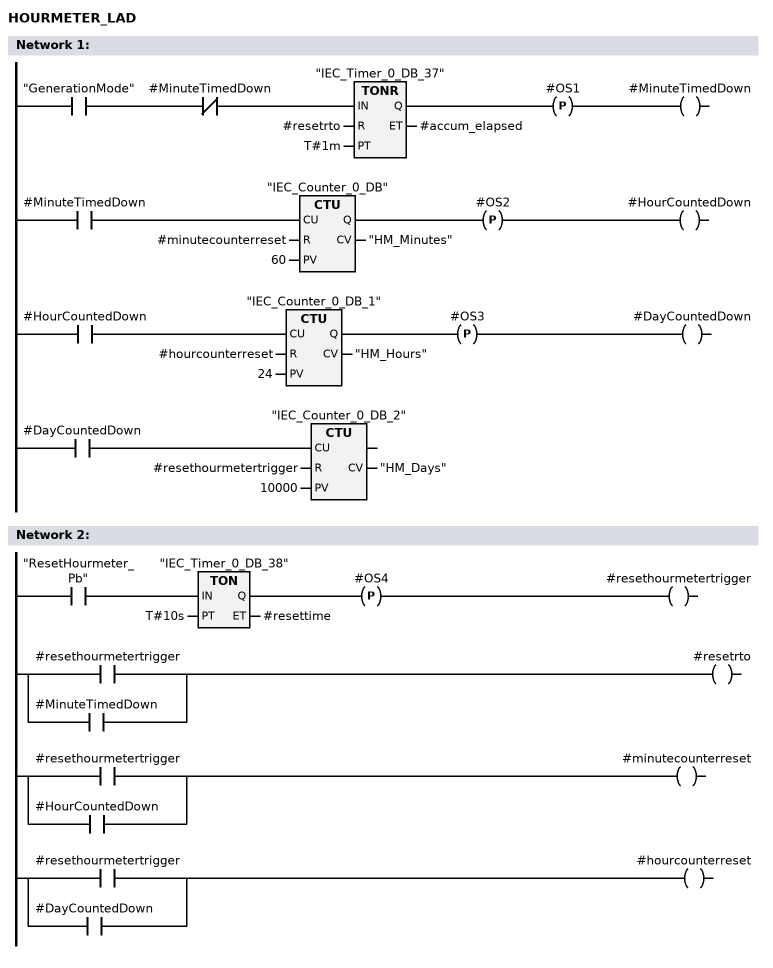
   "IEC_Timer_0_DB_37".TONR(IN := "GenerationMode" AND NOT #MinuteTimedDown,
                           R := #resetrto,
                           PT := T#1m,
                           ET => #accum_elapsed);
   #_w1 := "IEC_Timer_0_DB_37".Q AND NOT #OS1;   // rising edge
   #OS1 := "IEC_Timer_0_DB_37".Q;
   #MinuteTimedDown := #_w1;
   "IEC_Counter_0_DB".CTU(CU := #MinuteTimedDown, R := #minutecounterreset, PV := 60, CV => "HM_Minutes");
   #_w2 := "IEC_Counter_0_DB".Q AND NOT #OS2;   // rising edge
   #OS2 := "IEC_Counter_0_DB".Q;
   #HourCountedDown := #_w2;
   "IEC_Counter_0_DB_1".CTU(CU := #HourCountedDown, R := #hourcounterreset, PV := 24, CV => "HM_Hours");
   #_w3 := "IEC_Counter_0_DB_1".Q AND NOT #OS3;   // rising edge
   #OS3 := "IEC_Counter_0_DB_1".Q;
   #DayCountedDown := #_w3;
   "IEC_Counter_0_DB_2".CTU(CU := #DayCountedDown, R := #resethourmetertrigger, PV := 10000, CV => "HM_Days");
END_REGION

REGION Network 2
   "IEC_Timer_0_DB_38".TON(IN := "ResetHourmeter_Pb", PT := T#10s, ET => #resettime);
   #_w1 := "IEC_Timer_0_DB_38".Q AND NOT #OS4;   // rising edge
   #OS4 := "IEC_Timer_0_DB_38".Q;
   #resethourmetertrigger := #_w1;
   #resetrto := #resethourmetertrigger OR #MinuteTimedDown;
   #minutecounterreset := #resethourmetertrigger OR #HourCountedDown;
   #hourcounterreset := #resethourmetertrigger OR #DayCountedDown;
END_REGION
END_FUNCTION_BLOCK

FUNCTION_BLOCK "HOURMETER_FBD"   // FB20, FBD
{ S7_Optimized_Access := 'TRUE' }
VERSION : 0.1
   VAR
      OS1 : Bool;
      OS2 : Bool;
      OS3 : Bool;
      OS4 : Bool;
      rtotimerreset : Bool;
      minutecounterreset : Bool;
      hourcounterreset : Bool;
      hourmeterresettrigger : Bool;
      accumulatedtime : Time;
      minutetimeddown : Bool;
      hourcounteddown : Bool;
      daycounteddown : Bool;
   END_VAR
   VAR_TEMP   // added for the SCL form of the ladder/FBD networks
      _w1 : Bool;
      _w2 : Bool;
      _w3 : Bool;
   END_VAR
BEGIN

REGION Network 1
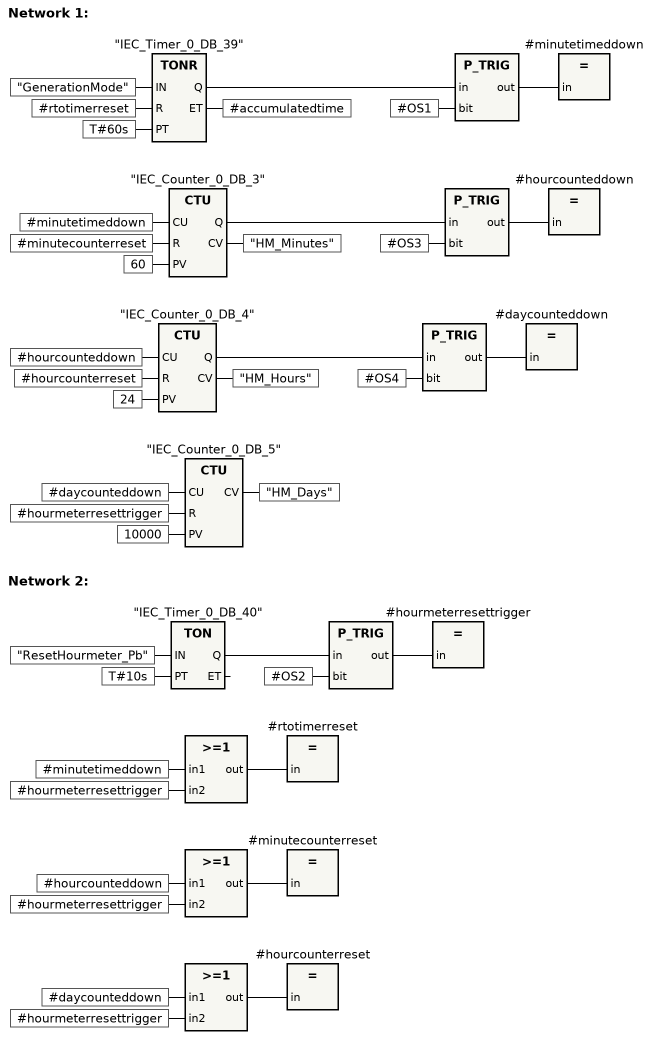
   "IEC_Timer_0_DB_39".TONR(IN := "GenerationMode", R := #rtotimerreset, PT := T#60s, ET => #accumulatedtime);
   #_w1 := "IEC_Timer_0_DB_39".Q AND NOT #OS1;   // rising edge
   #OS1 := "IEC_Timer_0_DB_39".Q;
   #minutetimeddown := #_w1;
   "IEC_Counter_0_DB_3".CTU(CU := #minutetimeddown, R := #minutecounterreset, PV := 60, CV => "HM_Minutes");
   #_w2 := "IEC_Counter_0_DB_3".Q AND NOT #OS3;   // rising edge
   #OS3 := "IEC_Counter_0_DB_3".Q;
   #hourcounteddown := #_w2;
   "IEC_Counter_0_DB_4".CTU(CU := #hourcounteddown, R := #hourcounterreset, PV := 24, CV => "HM_Hours");
   #_w3 := "IEC_Counter_0_DB_4".Q AND NOT #OS4;   // rising edge
   #OS4 := "IEC_Counter_0_DB_4".Q;
   #daycounteddown := #_w3;
   "IEC_Counter_0_DB_5".CTU(CU := #daycounteddown, R := #hourmeterresettrigger, PV := 10000, CV => "HM_Days");
END_REGION

REGION Network 2
   "IEC_Timer_0_DB_40".TON(IN := "ResetHourmeter_Pb", PT := T#10s);
   #_w1 := "IEC_Timer_0_DB_40".Q AND NOT #OS2;   // rising edge
   #OS2 := "IEC_Timer_0_DB_40".Q;
   #hourmeterresettrigger := #_w1;
   #rtotimerreset := #minutetimeddown OR #hourmeterresettrigger;
   #minutecounterreset := #hourcounteddown OR #hourmeterresettrigger;
   #hourcounterreset := #daycounteddown OR #hourmeterresettrigger;
END_REGION
END_FUNCTION_BLOCK

FUNCTION_BLOCK "HOURMETER_SCL"   // FB21, SCL
{ S7_Optimized_Access := 'TRUE' }
VERSION : 0.1
   VAR
      rtotimerreset : Bool;
      minutecounterreset : Bool;
      hourcounterreset : Bool;
      hourmeterresettrigger : Bool;
      accumulatedtime : Time;
      minutetimeddown : Bool;
      hourcounteddown : Bool;
      daycounteddown : Bool;
   END_VAR
BEGIN
   IF "GenerationMode" THEN
       "IEC_Timer_0_DB_41".TONR(IN := TRUE,
                                R := #rtotimerreset,
                                PT := T#60s,
                                Q => #minutetimeddown,
                                ET => #accumulatedtime);
   END_IF;

   IF #minutetimeddown THEN
       RESET_TIMER("IEC_Timer_0_DB_41");
   END_IF;

   "IEC_Counter_0_DB_6".CTU(CU:=#minutetimeddown,
                            R:=#minutecounterreset,
                            PV:=60,
                            Q=>#hourcounteddown,
                            CV=>"HM_Minutes");

   "IEC_Counter_0_DB_7".CTU(CU:=#hourcounteddown,
                            R:=#hourcounterreset,
                            PV:=24,
                            Q=>#daycounteddown,
                            CV=>"HM_Hours");

   "IEC_Counter_0_DB_9".CTU(CU:=#daycounteddown,
                            R:=#hourmeterresettrigger,
                            PV:=10000,
                            CV=>"HM_Days");

   IF "ResetHourmeter_Pb" THEN
       "IEC_Timer_0_DB_42".TON(IN:=TRUE,
                               PT:=T#10s,
                               Q=>#hourmeterresettrigger);
   ELSE
       RESET_TIMER("IEC_Timer_0_DB_42");
   END_IF;

   IF #hourmeterresettrigger OR #minutetimeddown THEN
       #rtotimerreset := 1;
   ELSE
       #rtotimerreset := 0;
   END_IF;

   IF #hourmeterresettrigger OR #hourcounteddown THEN
       #minutecounterreset := 1;
   ELSE
       #minutecounterreset := 0;
   END_IF;

   IF #hourmeterresettrigger OR #daycounteddown THEN
       #hourcounterreset := 1;
   ELSE
       #hourcounterreset := 0;
   END_IF;
END_FUNCTION_BLOCK

FUNCTION_BLOCK "HOURMETER_STL"   // FB22, STL
{ S7_Optimized_Access := 'TRUE' }
VERSION : 0.1
   VAR
      hourmeterresettrigger : Bool;
      minutecounterreset : Bool;
      hourcounterreset : Bool;
      minutetimeddown : Bool;
      hourcounteddown : Bool;
      daycounteddown : Bool;
      accumulatedtime : Time;
      rtotimerreset : Bool;
   END_VAR
   VAR_TEMP
      toomanydays : Bool;
      acctime : Time;
   END_VAR
BEGIN

REGION Network 1
         A     "GenerationMode";
         JC    RTOtimer;
         CLR;
         JU    EndOfLine;

   RTOtimer:CALL  TONR, "IEC_Timer_0_DB_43"
         ( IN := TRUE,
           R  := #rtotimerreset,
           PT := T#1m,
           Q  := #minutetimeddown,
           ET := #accumulatedtime
         );

         CALL  CTU, "IEC_Counter_0_DB_10"
         ( CU := #minutetimeddown,
           R  := #minutecounterreset,
           PV := 60,
           Q  := #hourcounteddown,
           CV := "HM_Minutes"
         );

         CALL  CTU, "IEC_Counter_0_DB_11"
         ( CU := #hourcounteddown,
           R  := #hourcounterreset,
           PV := 24,
           Q  := #daycounteddown,
           CV := "HM_Hours"
         );

         CALL  CTU, "IEC_Counter_0_DB_12"
         ( CU := #daycounteddown,
           R  := #hourmeterresettrigger,
           PV := 10000,
           Q  := #toomanydays,
           CV := "HM_Days"
         );

         JU    ResetEvaluate;

   ResetEvaluate:CLR;
         A     "ResetHourmeter_Pb";
         JC    ResetHourmeter;
         CALL  RESET_TIMER
         ( "TIMER" := "IEC_Timer_0_DB_44"
         );
         JU    EndOfLine;

   ResetHourmeter:CALL  TON, "IEC_Timer_0_DB_44"
         ( IN := TRUE,
           PT := T#10s,
           Q  := #hourmeterresettrigger,
           ET := #acctime
         );


   EndOfLine:A     #hourmeterresettrigger;
         O     #minutetimeddown;
         =     #rtotimerreset;
         CLR;
         A     #hourmeterresettrigger;
         O     #hourcounteddown;
         =     #minutecounterreset;
         CLR;
         A     #hourmeterresettrigger;
         O     #daycounteddown;
         =     #hourcounterreset;
         CLR;
         NOT;
         R     #hourmeterresettrigger;
END_REGION
END_FUNCTION_BLOCK

FUNCTION "SCP" : Void   // FC1, FBD
{ S7_Optimized_Access := 'TRUE' }
VERSION : 0.1
   VAR_INPUT
      Input_Min : Int;
      Input_Signal : Int;
      Input_Max : Int;
      Output_Min : Int;
      Output_Max : Int;
   END_VAR
   VAR_OUTPUT
      SV : Int;
   END_VAR
   VAR_TEMP
      tv : Real;
   END_VAR
BEGIN

REGION Network 1
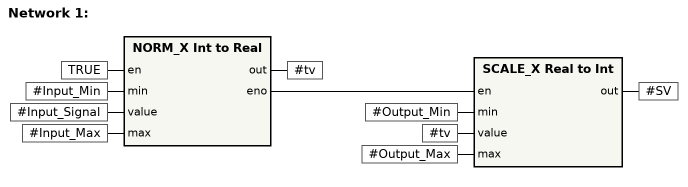
   IF TRUE THEN
       #tv := NORM_X(MIN := #Input_Min, VALUE := #Input_Signal, MAX := #Input_Max);
       #SV := SCALE_X(MIN := #Output_Min, VALUE := #tv, MAX := #Output_Max);
   END_IF;
END_REGION
END_FUNCTION

FUNCTION "CONVERTTIME" : Void   // FC2, FBD
{ S7_Optimized_Access := 'TRUE' }
VERSION : 0.1
   VAR_INPUT
      Int1 : Int;
   END_VAR
   VAR_OUTPUT
      Time1 : Time;
   END_VAR
   VAR_TEMP
      tv : Int;
   END_VAR
BEGIN

REGION Network 1
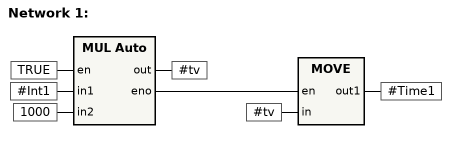
   IF TRUE THEN
       #tv := #Int1 * 1000;
       #Time1 := #tv;
   END_IF;
END_REGION
END_FUNCTION

ORGANIZATION_BLOCK "Main"   // OB1, LAD, ProgramCycle
TITLE = "Main Program Sweep (Cycle)"
{ S7_Optimized_Access := 'TRUE' }
VERSION : 0.1
   VAR_INPUT
      Initial_Call : Bool;   // Initial call of this OB
      Remanence : Bool;   // =True, if remanent data are available
   END_VAR
   VAR_TEMP
      SequenceInit : Bool;
      InitSequence : Bool;
   END_VAR
   VAR_TEMP   // added for the SCL form of the ladder/FBD networks
      _w1 : Bool;
      _w2 : Bool;
      _w3 : Bool;
      _w4 : Bool;
   END_VAR
BEGIN

REGION Network 1
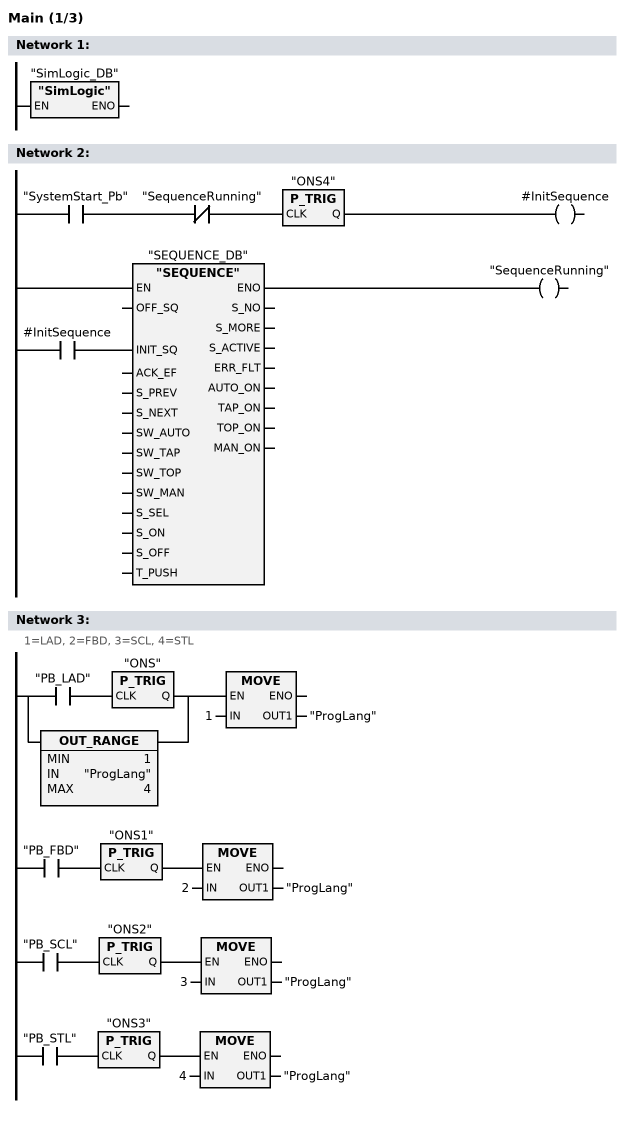
   RUNG wire#powerrail
      "SimLogic_DB"()
   END_RUNG
   // the same network as SCL:
   "SimLogic_DB"();   // "SimLogic"
END_REGION

REGION Network 2
   RUNG wire#powerrail
      Contact( "SystemStart_Pb" )
      I_Contact( "SequenceRunning" )
      P_Trig( "ONS4" )
      Coil( #InitSequence )
   END_RUNG
   RUNG wire#powerrail
      "SEQUENCE_DB"(INIT_SQ := wire#w1, OFF_SQ :=, ACK_EF :=, S_PREV :=, S_NEXT :=, SW_AUTO :=, SW_TAP :=, SW_TOP :=, SW_MAN :=, S_SEL :=, S_ON :=, S_OFF :=, T_PUSH :=, S_NO =>, S_MORE =>, S_ACTIVE =>, ERR_FLT =>, AUTO_ON =>, TAP_ON =>, TOP_ON =>, MAN_ON =>)
      Coil( "SequenceRunning" )
   END_RUNG
   RUNG wire#powerrail
      Contact( #InitSequence )
   END_RUNG wire#w1
   // the same network as SCL:
   #_w1 := "SystemStart_Pb" AND NOT "SequenceRunning";
   #_w2 := #_w1 AND NOT "ONS4";   // rising edge
   "ONS4" := #_w1;
   #InitSequence := #_w2;
   "SEQUENCE_DB"(INIT_SQ := #InitSequence, ENO => #_w3);   // "SEQUENCE"
   "SequenceRunning" := #_w3;
END_REGION

REGION Network 3
   // 1=LAD, 2=FBD, 3=SCL, 4=STL
   #_w1 := "PB_LAD" AND NOT "ONS";   // rising edge
   "ONS" := "PB_LAD";
   IF #_w1 OR ("ProgLang" < 1) OR ("ProgLang" > 4) THEN "ProgLang" := 1; END_IF;
   #_w2 := "PB_FBD" AND NOT "ONS1";   // rising edge
   "ONS1" := "PB_FBD";
   IF #_w2 THEN "ProgLang" := 2; END_IF;
   #_w3 := "PB_SCL" AND NOT "ONS2";   // rising edge
   "ONS2" := "PB_SCL";
   IF #_w3 THEN "ProgLang" := 3; END_IF;
   #_w4 := "PB_STL" AND NOT "ONS3";   // rising edge
   "ONS3" := "PB_STL";
   IF #_w4 THEN "ProgLang" := 4; END_IF;
END_REGION

REGION Network 4
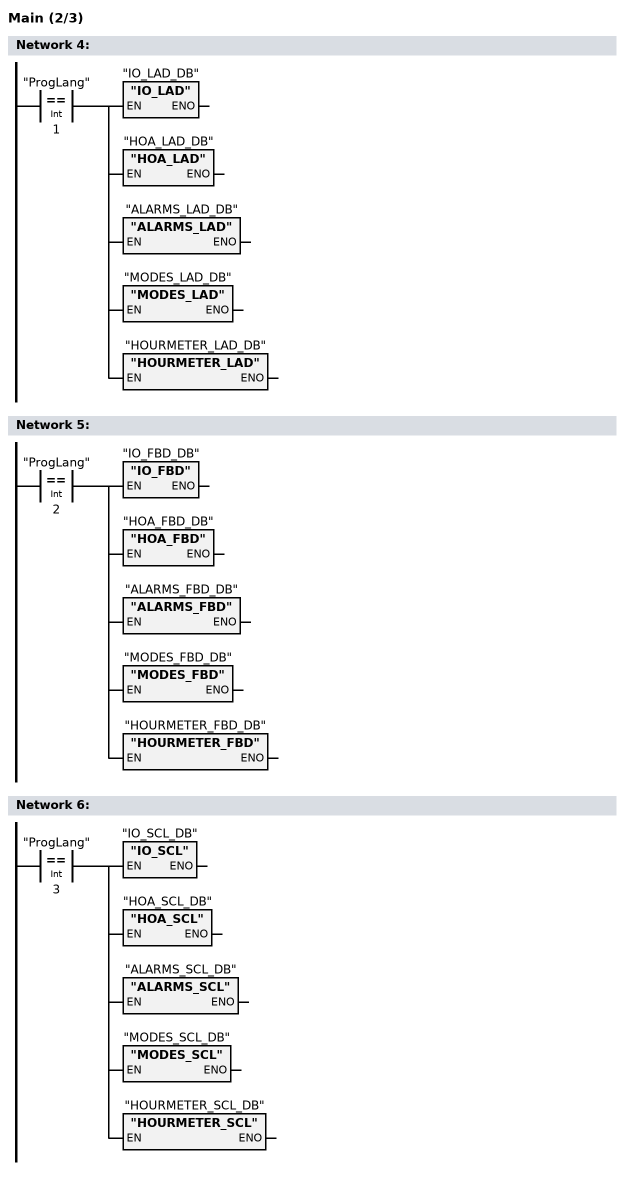
   RUNG wire#powerrail
      { S7_Templates := "SrcType := Int" } EQ_Contact(in1 := "ProgLang", in2 := 1)
      wire#w1
      "IO_LAD_DB"()
   END_RUNG
   RUNG wire#w1
      "HOA_LAD_DB"()
   END_RUNG
   RUNG wire#w1
      "ALARMS_LAD_DB"()
   END_RUNG
   RUNG wire#w1
      "MODES_LAD_DB"()
   END_RUNG
   RUNG wire#w1
      "HOURMETER_LAD_DB"()
   END_RUNG
   // the same network as SCL:
   #_w1 := "ProgLang" = 1;
   IF #_w1 THEN
       "IO_LAD_DB"();   // "IO_LAD"
       "HOA_LAD_DB"();   // "HOA_LAD"
       "ALARMS_LAD_DB"();   // "ALARMS_LAD"
       "MODES_LAD_DB"();   // "MODES_LAD"
       "HOURMETER_LAD_DB"();   // "HOURMETER_LAD"
   END_IF;
END_REGION

REGION Network 5
   RUNG wire#powerrail
      { S7_Templates := "SrcType := Int" } EQ_Contact(in1 := "ProgLang", in2 := 2)
      wire#w1
      "IO_FBD_DB"()
   END_RUNG
   RUNG wire#w1
      "HOA_FBD_DB"()
   END_RUNG
   RUNG wire#w1
      "ALARMS_FBD_DB"()
   END_RUNG
   RUNG wire#w1
      "MODES_FBD_DB"()
   END_RUNG
   RUNG wire#w1
      "HOURMETER_FBD_DB"()
   END_RUNG
   // the same network as SCL:
   #_w1 := "ProgLang" = 2;
   IF #_w1 THEN
       "IO_FBD_DB"();   // "IO_FBD"
       "HOA_FBD_DB"();   // "HOA_FBD"
       "ALARMS_FBD_DB"();   // "ALARMS_FBD"
       "MODES_FBD_DB"();   // "MODES_FBD"
       "HOURMETER_FBD_DB"();   // "HOURMETER_FBD"
   END_IF;
END_REGION

REGION Network 6
   RUNG wire#powerrail
      { S7_Templates := "SrcType := Int" } EQ_Contact(in1 := "ProgLang", in2 := 3)
      wire#w1
      "IO_SCL_DB"()
   END_RUNG
   RUNG wire#w1
      "HOA_SCL_DB"()
   END_RUNG
   RUNG wire#w1
      "ALARMS_SCL_DB"()
   END_RUNG
   RUNG wire#w1
      "MODES_SCL_DB"()
   END_RUNG
   RUNG wire#w1
      "HOURMETER_SCL_DB"()
   END_RUNG
   // the same network as SCL:
   #_w1 := "ProgLang" = 3;
   IF #_w1 THEN
       "IO_SCL_DB"();   // "IO_SCL"
       "HOA_SCL_DB"();   // "HOA_SCL"
       "ALARMS_SCL_DB"();   // "ALARMS_SCL"
       "MODES_SCL_DB"();   // "MODES_SCL"
       "HOURMETER_SCL_DB"();   // "HOURMETER_SCL"
   END_IF;
END_REGION

REGION Network 7
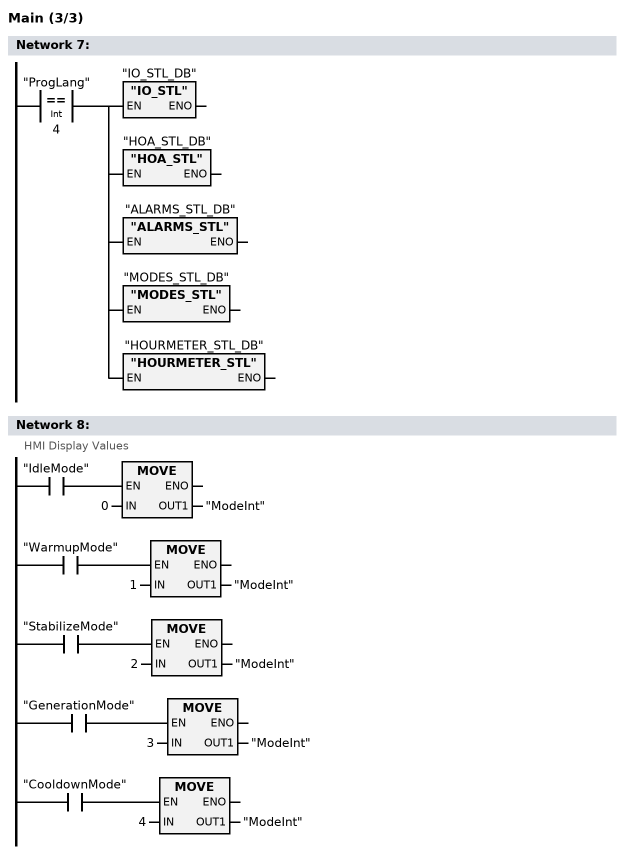
   RUNG wire#powerrail
      { S7_Templates := "SrcType := Int" } EQ_Contact(in1 := "ProgLang", in2 := 4)
      wire#w1
      "IO_STL_DB"()
   END_RUNG
   RUNG wire#w1
      "HOA_STL_DB"()
   END_RUNG
   RUNG wire#w1
      "ALARMS_STL_DB"()
   END_RUNG
   RUNG wire#w1
      "MODES_STL_DB"()
   END_RUNG
   RUNG wire#w1
      "HOURMETER_STL_DB"()
   END_RUNG
   // the same network as SCL:
   #_w1 := "ProgLang" = 4;
   IF #_w1 THEN
       "IO_STL_DB"();   // "IO_STL"
       "HOA_STL_DB"();   // "HOA_STL"
       "ALARMS_STL_DB"();   // "ALARMS_STL"
       "MODES_STL_DB"();   // "MODES_STL"
       "HOURMETER_STL_DB"();   // "HOURMETER_STL"
   END_IF;
END_REGION

REGION Network 8
   // HMI Display Values
   RUNG wire#powerrail
      Contact( "IdleMode" )
      Move(in := 0, out1 => "ModeInt")
   END_RUNG
   RUNG wire#powerrail
      Contact( "WarmupMode" )
      Move(in := 1, out1 => "ModeInt")
   END_RUNG
   RUNG wire#powerrail
      Contact( "StabilizeMode" )
      Move(in := 2, out1 => "ModeInt")
   END_RUNG
   RUNG wire#powerrail
      Contact( "GenerationMode" )
      Move(in := 3, out1 => "ModeInt")
   END_RUNG
   RUNG wire#powerrail
      Contact( "CooldownMode" )
      Move(in := 4, out1 => "ModeInt")
   END_RUNG
   // the same network as SCL:
   IF "IdleMode" THEN "ModeInt" := 0; END_IF;
   IF "WarmupMode" THEN "ModeInt" := 1; END_IF;
   IF "StabilizeMode" THEN "ModeInt" := 2; END_IF;
   IF "GenerationMode" THEN "ModeInt" := 3; END_IF;
   IF "CooldownMode" THEN "ModeInt" := 4; END_IF;
END_REGION
END_ORGANIZATION_BLOCK

ORGANIZATION_BLOCK "PID"   // OB31, LAD, CyclicInterrupt
{ S7_Optimized_Access := 'TRUE' }
VERSION : 0.1
   VAR_INPUT
      Initial_Call : Bool;   // Initial call of this OB
      Event_Count : Int;   // Events discarded
   END_VAR
   VAR_TEMP
      Bsp : Real;
      Vsp : Real;
      BaffleHandTrigger : Bool;
      BaffleOffTrigger : Bool;
      VFDHandTrigger : Bool;
      VFDOffTrigger : Bool;
      BaffleAutoTrigger : Bool;
      VFDautoTrigger : Bool;
   END_VAR
   VAR_TEMP   // added for the SCL form of the ladder/FBD networks
      _w1 : Bool;
      _w2 : Bool;
      _w3 : Bool;
      _w4 : Bool;
      _w5 : Bool;
      _w6 : Bool;
      _w7 : Bool;
   END_VAR
BEGIN

REGION Network 1
   // High Oil Flow Alarm Handling
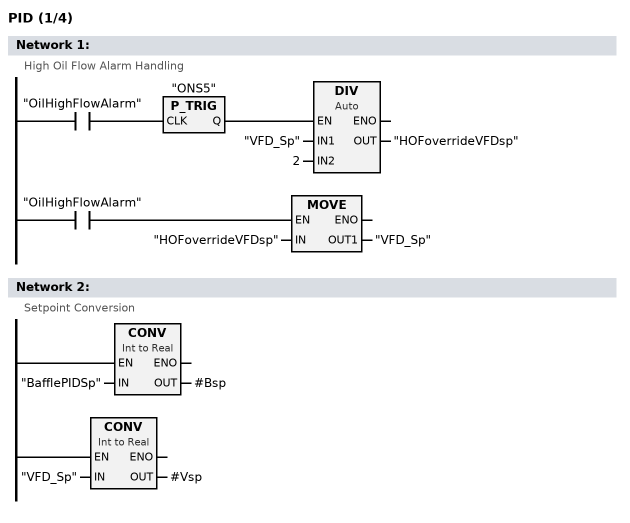
   RUNG wire#powerrail
      Contact( "OilHighFlowAlarm" )
      P_Trig( "ONS5" )
      Div(in1 := "VFD_Sp", in2 := 2, out => "HOFoverrideVFDsp")
   END_RUNG
   RUNG wire#powerrail
      Contact( "OilHighFlowAlarm" )
      Move(in := "HOFoverrideVFDsp", out1 => "VFD_Sp")
   END_RUNG
   // the same network as SCL:
   #_w1 := "OilHighFlowAlarm" AND NOT "ONS5";   // rising edge
   "ONS5" := "OilHighFlowAlarm";
   IF #_w1 THEN "HOFoverrideVFDsp" := "VFD_Sp" / 2; END_IF;
   IF "OilHighFlowAlarm" THEN "VFD_Sp" := "HOFoverrideVFDsp"; END_IF;
END_REGION

REGION Network 2
   // Setpoint Conversion
   RUNG wire#powerrail
      { S7_Templates := "[SrcType := Int, DestType := Real]" } Convert(in := "BafflePIDSp", out => #Bsp)
   END_RUNG
   RUNG wire#powerrail
      { S7_Templates := "[SrcType := Int, DestType := Real]" } Convert(in := "VFD_Sp", out => #Vsp)
   END_RUNG
   // the same network as SCL:
   #Bsp := INT_TO_REAL("BafflePIDSp");
   #Vsp := INT_TO_REAL("VFD_Sp");
END_REGION

REGION Network 3
   // Baffle HOA
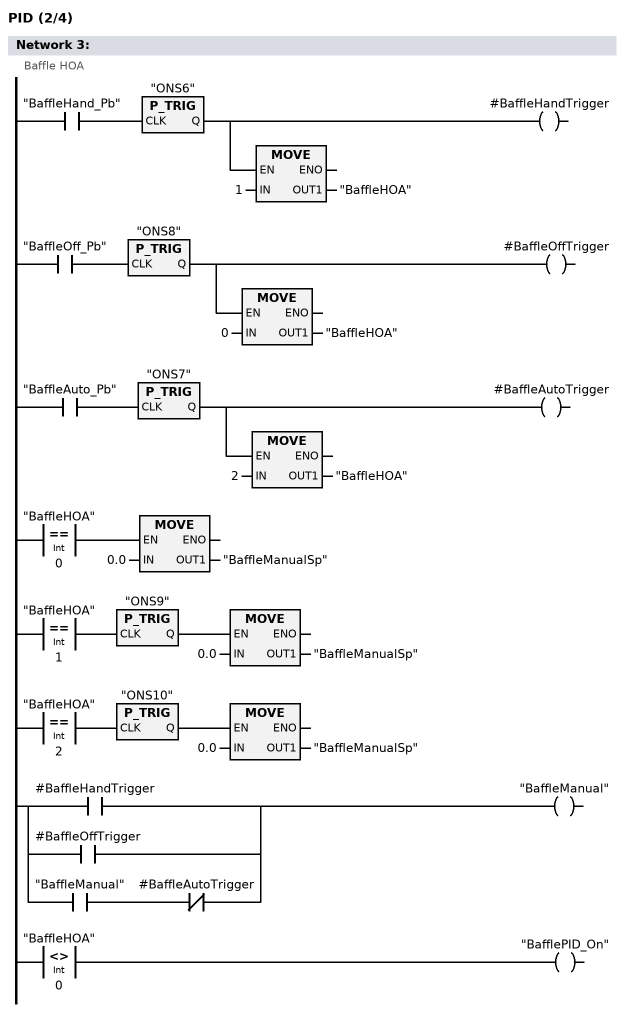
   RUNG wire#powerrail
      Contact( "BaffleHand_Pb" )
      P_Trig( "ONS6" )
      wire#w1
      Coil( #BaffleHandTrigger )
   END_RUNG
   RUNG wire#w1
      Move(in := 1, out1 => "BaffleHOA")
   END_RUNG
   RUNG wire#powerrail
      Contact( "BaffleOff_Pb" )
      P_Trig( "ONS8" )
      wire#w2
      Coil( #BaffleOffTrigger )
   END_RUNG
   RUNG wire#w2
      Move(in := 0, out1 => "BaffleHOA")
   END_RUNG
   RUNG wire#powerrail
      Contact( "BaffleAuto_Pb" )
      P_Trig( "ONS7" )
      wire#w3
      Coil( #BaffleAutoTrigger )
   END_RUNG
   RUNG wire#w3
      Move(in := 2, out1 => "BaffleHOA")
   END_RUNG
   RUNG wire#powerrail
      { S7_Templates := "SrcType := Int" } EQ_Contact(in1 := "BaffleHOA", in2 := 0)
      Move(in := 0.0, out1 => "BaffleManualSp")
   END_RUNG
   RUNG wire#powerrail
      { S7_Templates := "SrcType := Int" } EQ_Contact(in1 := "BaffleHOA", in2 := 1)
      P_Trig( "ONS9" )
      Move(in := 0.0, out1 => "BaffleManualSp")
   END_RUNG
   RUNG wire#powerrail
      { S7_Templates := "SrcType := Int" } EQ_Contact(in1 := "BaffleHOA", in2 := 2)
      P_Trig( "ONS10" )
      Move(in := 0.0, out1 => "BaffleManualSp")
   END_RUNG
   RUNG wire#powerrail
      Contact( #BaffleHandTrigger )
      wire#w4
      Coil( "BaffleManual" )
   END_RUNG
   RUNG wire#powerrail
      Contact( #BaffleOffTrigger )
   END_RUNG wire#w4
   RUNG wire#powerrail
      Contact( "BaffleManual" )
      I_Contact( #BaffleAutoTrigger )
   END_RUNG wire#w4
   RUNG wire#powerrail
      { S7_Templates := "SrcType := Int" } NE_Contact(in1 := "BaffleHOA", in2 := 0)
      Coil( "BafflePID_On" )
   END_RUNG
   // the same network as SCL:
   #_w1 := "BaffleHand_Pb" AND NOT "ONS6";   // rising edge
   "ONS6" := "BaffleHand_Pb";
   #BaffleHandTrigger := #_w1;
   IF #_w1 THEN "BaffleHOA" := 1; END_IF;
   #_w2 := "BaffleOff_Pb" AND NOT "ONS8";   // rising edge
   "ONS8" := "BaffleOff_Pb";
   #BaffleOffTrigger := #_w2;
   IF #_w2 THEN "BaffleHOA" := 0; END_IF;
   #_w3 := "BaffleAuto_Pb" AND NOT "ONS7";   // rising edge
   "ONS7" := "BaffleAuto_Pb";
   #BaffleAutoTrigger := #_w3;
   IF #_w3 THEN "BaffleHOA" := 2; END_IF;
   IF "BaffleHOA" = 0 THEN "BaffleManualSp" := 0.0; END_IF;
   #_w4 := "BaffleHOA" = 1;
   #_w5 := #_w4 AND NOT "ONS9";   // rising edge
   "ONS9" := #_w4;
   IF #_w5 THEN "BaffleManualSp" := 0.0; END_IF;
   #_w6 := "BaffleHOA" = 2;
   #_w7 := #_w6 AND NOT "ONS10";   // rising edge
   "ONS10" := #_w6;
   IF #_w7 THEN "BaffleManualSp" := 0.0; END_IF;
   "BaffleManual" := #BaffleHandTrigger OR #BaffleOffTrigger OR ("BaffleManual" AND NOT #BaffleAutoTrigger);
   "BafflePID_On" := "BaffleHOA" <> 0;
END_REGION

REGION Network 4
   // VFD HOA
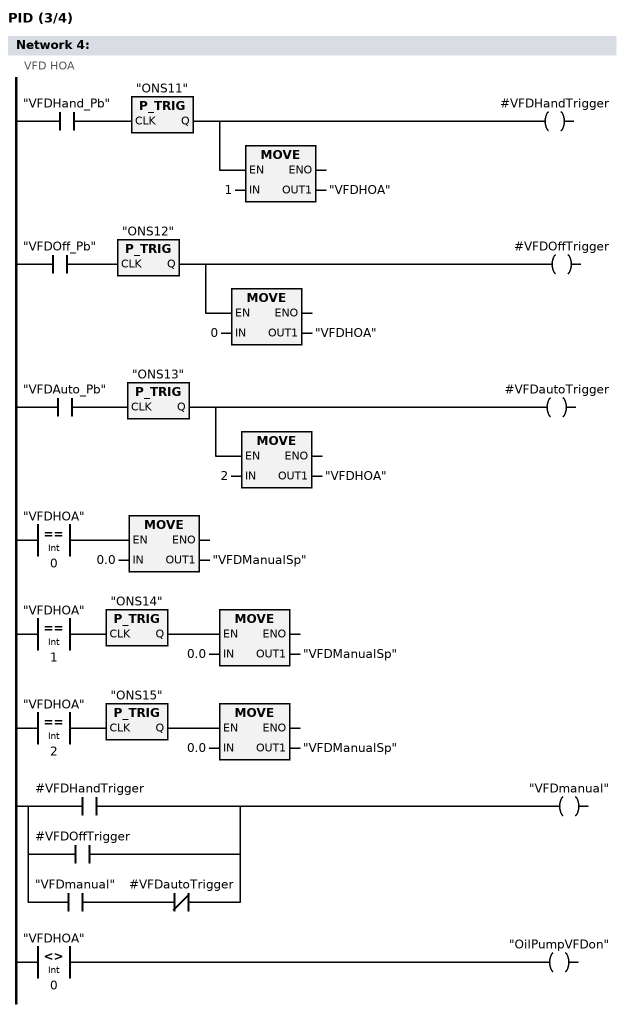
   RUNG wire#powerrail
      Contact( "VFDHand_Pb" )
      P_Trig( "ONS11" )
      wire#w1
      Coil( #VFDHandTrigger )
   END_RUNG
   RUNG wire#w1
      Move(in := 1, out1 => "VFDHOA")
   END_RUNG
   RUNG wire#powerrail
      Contact( "VFDOff_Pb" )
      P_Trig( "ONS12" )
      wire#w2
      Coil( #VFDOffTrigger )
   END_RUNG
   RUNG wire#w2
      Move(in := 0, out1 => "VFDHOA")
   END_RUNG
   RUNG wire#powerrail
      Contact( "VFDAuto_Pb" )
      P_Trig( "ONS13" )
      wire#w3
      Coil( #VFDautoTrigger )
   END_RUNG
   RUNG wire#w3
      Move(in := 2, out1 => "VFDHOA")
   END_RUNG
   RUNG wire#powerrail
      { S7_Templates := "SrcType := Int" } EQ_Contact(in1 := "VFDHOA", in2 := 0)
      Move(in := 0.0, out1 => "VFDManualSp")
   END_RUNG
   RUNG wire#powerrail
      { S7_Templates := "SrcType := Int" } EQ_Contact(in1 := "VFDHOA", in2 := 1)
      P_Trig( "ONS14" )
      Move(in := 0.0, out1 => "VFDManualSp")
   END_RUNG
   RUNG wire#powerrail
      { S7_Templates := "SrcType := Int" } EQ_Contact(in1 := "VFDHOA", in2 := 2)
      P_Trig( "ONS15" )
      Move(in := 0.0, out1 => "VFDManualSp")
   END_RUNG
   RUNG wire#powerrail
      Contact( #VFDHandTrigger )
      wire#w4
      Coil( "VFDmanual" )
   END_RUNG
   RUNG wire#powerrail
      Contact( #VFDOffTrigger )
   END_RUNG wire#w4
   RUNG wire#powerrail
      Contact( "VFDmanual" )
      I_Contact( #VFDautoTrigger )
   END_RUNG wire#w4
   RUNG wire#powerrail
      { S7_Templates := "SrcType := Int" } NE_Contact(in1 := "VFDHOA", in2 := 0)
      Coil( "OilPumpVFDon" )
   END_RUNG
   // the same network as SCL:
   #_w1 := "VFDHand_Pb" AND NOT "ONS11";   // rising edge
   "ONS11" := "VFDHand_Pb";
   #VFDHandTrigger := #_w1;
   IF #_w1 THEN "VFDHOA" := 1; END_IF;
   #_w2 := "VFDOff_Pb" AND NOT "ONS12";   // rising edge
   "ONS12" := "VFDOff_Pb";
   #VFDOffTrigger := #_w2;
   IF #_w2 THEN "VFDHOA" := 0; END_IF;
   #_w3 := "VFDAuto_Pb" AND NOT "ONS13";   // rising edge
   "ONS13" := "VFDAuto_Pb";
   #VFDautoTrigger := #_w3;
   IF #_w3 THEN "VFDHOA" := 2; END_IF;
   IF "VFDHOA" = 0 THEN "VFDManualSp" := 0.0; END_IF;
   #_w4 := "VFDHOA" = 1;
   #_w5 := #_w4 AND NOT "ONS14";   // rising edge
   "ONS14" := #_w4;
   IF #_w5 THEN "VFDManualSp" := 0.0; END_IF;
   #_w6 := "VFDHOA" = 2;
   #_w7 := #_w6 AND NOT "ONS15";   // rising edge
   "ONS15" := #_w6;
   IF #_w7 THEN "VFDManualSp" := 0.0; END_IF;
   "VFDmanual" := #VFDHandTrigger OR #VFDOffTrigger OR ("VFDmanual" AND NOT #VFDautoTrigger);
   "OilPumpVFDon" := "VFDHOA" <> 0;
END_REGION

REGION Network 5
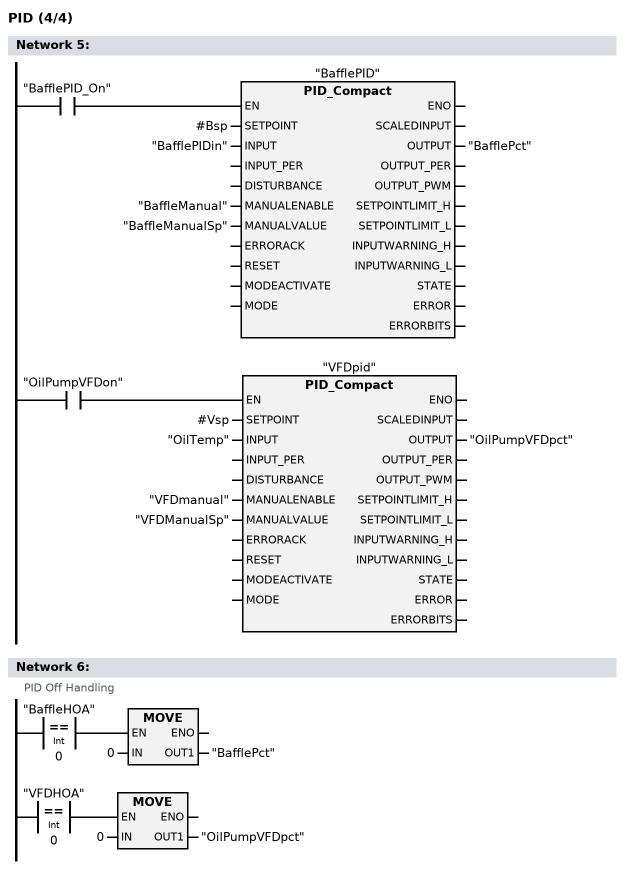
   IF "BafflePID_On" THEN
       "BafflePID"(Setpoint := #Bsp,   // PID_Compact
                   Input := "BafflePIDin",
                   ManualEnable := "BaffleManual",
                   ManualValue := "BaffleManualSp",
                   Output => "BafflePct");
   END_IF;
   IF "OilPumpVFDon" THEN
       "VFDpid"(Setpoint := #Vsp,   // PID_Compact
                Input := "OilTemp",
                ManualEnable := "VFDmanual",
                ManualValue := "VFDManualSp",
                Output => "OilPumpVFDpct");
   END_IF;
END_REGION

REGION Network 6
   // PID Off Handling
   RUNG wire#powerrail
      { S7_Templates := "SrcType := Int" } EQ_Contact(in1 := "BaffleHOA", in2 := 0)
      Move(in := 0, out1 => "BafflePct")
   END_RUNG
   RUNG wire#powerrail
      { S7_Templates := "SrcType := Int" } EQ_Contact(in1 := "VFDHOA", in2 := 0)
      Move(in := 0, out1 => "OilPumpVFDpct")
   END_RUNG
   // the same network as SCL:
   IF "BaffleHOA" = 0 THEN "BafflePct" := 0; END_IF;
   IF "VFDHOA" = 0 THEN "OilPumpVFDpct" := 0; END_IF;
END_REGION
END_ORGANIZATION_BLOCK

(* ===== HMI "HMI_RT_1" =====
system functions are stored by id; their names below are inferred from use
connection "1500PLC": S71200_TCP_IP, SCADA_S7_1500_OMS

HMI tags "Default tag table"
   "SystemStartPb" : Bool = PLC SystemStart_Pb AT %M65.2, 500 ms
   "SystemStopPb" : Bool = PLC SystemStop_Pb AT %M65.4, 500 ms
   "EStopAlarm" : Bool = PLC EStopAlarm AT %M49.3, 500 ms
   "BrakeFailureAlarm" : Bool = PLC BrakeFailureAlarm AT %M49.0, 500 ms
   "OverspeedAlarm" : Bool = PLC OverspeedAlarm AT %M48.4, 500 ms
   "OvercurrentAlarm" : Bool = PLC OvercurrentAlarm AT %M48.0, 500 ms
   "HighOilTempAlarm" : Bool = PLC HighOilTempAlarm AT %M48.2, 500 ms
   "HighOilFlowAlarm" : Bool = PLC OilHighFlowAlarm AT %M48.6, 500 ms
   "LowOilFlowAlarm" : Bool = PLC OilLowFlowAlarm AT %M5.6, 500 ms
   "AlarmSilence" : Bool = PLC AlarmSilence AT %M5.5, 500 ms
   "AlarmReset" : Bool = PLC AlarmReset AT %M5.4, 500 ms
   "BrakeEn" : Bool = PLC Brake_Out AT %M4.0, 500 ms
   "StationintlkEn" : Bool = PLC StationInterlock_Out AT %M3.1, 500 ms
   "VFDen" : Bool = PLC OilPumpVFDen_Out AT %M4.1, 500 ms
   "BaffleEn" : Int = PLC Baffle_Out AT %MW18, 500 ms
   "AlarmHornEn" : Bool = PLC AlarmHorn_Out AT %M3.0, 500 ms
   "BrakeHandPb" : Bool = PLC BrakeHand_Pb AT %M3.6, 500 ms
   "BrakeOffPb" : Bool = PLC BrakeOff_Pb AT %M3.5, 500 ms
   "BrakeAutoPb" : Bool = PLC BrakeAuto_Pb AT %M3.7, 500 ms
   "StationintlkHandPb" : Bool = PLC StationIntHand_Pb AT %M4.6, 500 ms
   "StationintlkOffPb" : Bool = PLC StationIntOff_Pb AT %M4.5, 500 ms
   "StationintlkAutoPb" : Bool = PLC StationIntAuto_Pb AT %M4.7, 500 ms
   "VFDhandPb" : Bool = PLC VFDHand_Pb AT %M99.3, 500 ms
   "VFDoffPb" : Bool = PLC VFDOff_Pb AT %M99.4, 500 ms
   "VFDautoPb" : Bool = PLC VFDAuto_Pb AT %M99.5, 500 ms
   "BaffleHandPb" : Bool = PLC BaffleHand_Pb AT %M98.5, 500 ms
   "BaffleOffPb" : Bool = PLC BaffleOff_Pb AT %M98.6, 500 ms
   "BaffleAutoPb" : Bool = PLC BaffleAuto_Pb AT %M98.4, 500 ms
   "AlarmHornHandPb" : Bool = PLC AlarmHornHand_Pb AT %M4.3, 500 ms
   "AlarmHornOffPb" : Bool = PLC AlarmHornOff_Pb AT %M4.2, 500 ms
   "AlarmHornAutoPb" : Bool = PLC AlarmHornAuto_Pb AT %M4.4, 500 ms
   "ModeInt" : Int = PLC ModeInt AT %MW118, 500 ms
   "BrakeHOA" : Int = PLC BrakeHoa AT %MW34, 500 ms
   "StationintlkHOA" : Int = PLC StationIntHoa AT %MW38, 500 ms
   "VFDhoa" : Int = PLC VFDHOA AT %MW108, 500 ms
   "BaffleHOA" : Int = PLC BaffleHOA AT %MW74, 500 ms
   "AlarmHornHOA" : Int = PLC AlarmHornHoa AT %MW36, 500 ms
   "HM_Minutes" : Int = PLC HM_Minutes AT %MW32, 500 ms
   "HM_Hours" : Int = PLC HM_Hours AT %MW114, 500 ms
   "HM_Days" : Int = PLC HM_Days AT %MW116, 500 ms
   "HM_ResetPb" : Bool = PLC ResetHourmeter_Pb AT %M106.7, 500 ms
   "FaultMode" : Bool = PLC FaultMode AT %M64.6, 500 ms
   "BrakeFailureDelay" : Int = PLC BrakeFailureDelay_Sp AT %MW62, 500 ms
   "OverCurrentSp" : Int = PLC OvercurrentSp AT %MW46, 500 ms
   "OvercurrentDelay" : Int = PLC OvercurrentDelay_Sp AT %MW44, 500 ms
   "OverspeedSp" : Int = PLC OverspeedSp AT %MW56, 500 ms
   "OverspeedDelay" : Int = PLC OverspeedDelay_Sp AT %MW54, 500 ms
   "HighOilTempSp" : Int = PLC HighOilTempSp AT %MW52, 500 ms
   "HighOilTempDelay" : Int = PLC HighOilTempDelay_Sp AT %MW50, 500 ms
   "HighOilFlowSp" : Int = PLC OilHHflowSp AT %MW60, 500 ms
   "HighOilFlowDelay" : Int = PLC OilHighFlowDelay_Sp AT %MW58, 500 ms
   "LowOilFlowSp" : Int = PLC OilLLflowSp AT %MW42, 500 ms
   "LowOilFlowDelay" : Int = PLC OilLowFlowDelay_Sp AT %MW40, 500 ms
   "WarmupOilTemp" : Int = PLC WarmupOilTemp AT %MW80, 500 ms
   "WarmUpDelay" : Int = PLC WarmupOilTempDelaySp AT %MW82, 500 ms
   "CurrentSp" : Int = PLC StabilizekWSp AT %MW86, 500 ms
   "StabilizeDelay" : Int = PLC StabilizeDelaySp AT %MW88, 500 ms
   "CooldownOilTemp" : Int = PLC CooldownOilTempSp AT %MW96, 500 ms
   "CooldownDelay" : Int = PLC CooldownDelaySp AT %MW92, 500 ms
   "VFDmanualSp" : Real = PLC VFDManualSp AT %MD110, 500 ms
   "BaffleManualSp" : Real = PLC BaffleManualSp AT %MD102, 500 ms
   "ProgramLanguage" : Int = PLC ProgLang AT %MW0, 500 ms
   "LADpb" : Bool = PLC PB_LAD AT %M2.1, 500 ms
   "FBDpb" : Bool = PLC PB_FBD AT %M2.5, 500 ms
   "SCLpb" : Bool = PLC PB_SCL AT %M2.6, 500 ms
   "STLpb" : Bool = PLC PB_STL AT %M2.7, 500 ms
   "Current" : Int = PLC Current AT %MW28, 500 ms
   "OilTemp" : Int = PLC OilTemp AT %MW20, 500 ms
   "OilFlow" : Int = PLC OilFlow AT %MW22, 500 ms
   "BafflePct" : Int = PLC BafflePct AT %MW10, 500 ms
   "VFDpct" : Int = PLC OilPumpVFDpct AT %MW8, 500 ms
   "RPM" : Int = PLC RPM AT %MW26, 500 ms
   "EStopNotify" : Bool = PLC EStopNotify AT %M49.4, 500 ms
   "BrakFailureNotify" : Bool = PLC BrakeFailureNotify AT %M49.1, 500 ms
   "OverspeedNotify" : Bool = PLC OverspeedNotify AT %M48.5, 500 ms
   "OvercurrentNotify" : Bool = PLC OvercurrentNotify AT %M48.1, 500 ms
   "HiTempNotify" : Bool = PLC HighOilTempNotify AT %M48.3, 500 ms
   "LoFlowNotify" : Bool = PLC OilLowFlowNotify AT %M5.7, 500 ms
   "HiFlowNotify" : Bool = PLC OilHighFlowNotify AT %M48.7, 500 ms

discrete alarms
   1: 'Estop open', class Errors, trigger "EStopNotify" bit 0
   2: 'Brake failed', class Errors, trigger "BrakFailureNotify" bit 0
   3: 'Overcurrent', class Errors, trigger "OvercurrentNotify" bit 0
   4: 'Overspeed', class Errors, trigger "OverspeedNotify" bit 0
   5: 'Hi oil flow', class Errors, trigger "HiFlowNotify" bit 0
   6: 'Lo oil flow', class Errors, trigger "LoFlowNotify" bit 0
   7: 'Hi oil temp', class Errors, trigger "HiTempNotify" bit 0

screen "Status" 500x500
   TextField "Text field_17" at 190,223 size 81x30; Text 'OFFLINE'
      Visibility <- "StationintlkEn"
   Button "Button_1" at 13,455 size 80x30; TextOff 'Main'
      on Click: ActivateScreen("Status", 0)
   Button "Button_2" at 109,455 size 80x30; TextOff 'Overview'
      on Click: ActivateScreen("Overview", 0)
   Button "Button_3" at 205,455 size 80x30; TextOff 'Alarms'
      on Click: ActivateScreen("Alarms", 0)
   Button "Button_4" at 301,455 size 80x30; TextOff 'Config'
      on Click: ActivateScreen("Config", 0)
   TextField "Text field_3" at 8,8 size 155x30; Text 'System Status'
   TextField "Text field_4" at 349,50 size 134x38; Text 'Idle Mode'
      Visibility <- "ModeInt"
   TextField "Text field_5" at 287,50 size 196x38; Text 'Warmup Mode'
      Visibility <- "ModeInt"
   TextField "Text field_6" at 290,50 size 193x38; Text 'Stabilize Mode'
      Visibility <- "ModeInt"
   TextField "Text field_7" at 254,50 size 229x38; Text 'Generation Mode'
      Visibility <- "ModeInt"
   TextField "Text field_8" at 273,50 size 212x38; Text 'Cooldown Mode'
      Visibility <- "ModeInt"
   TextField "Text field_9" at 322,295 size 145x26; Text 'Ladder Diagram'
      Visibility <- "ProgramLanguage"
   RoundButton "Round button_1" at 336,329 size 48x48; Text 'LAD'
      on PressLeft: SetBit("LADpb")
      on ReleaseLeft: ResetBit("LADpb")
   RoundButton "Round button_2" at 386,329 size 48x48; Text 'FBD'
      on PressLeft: SetBit("FBDpb")
      on ReleaseLeft: ResetBit("FBDpb")
   RoundButton "Round button_3" at 336,381 size 48x48; Text 'SCL'
      on PressLeft: SetBit("SCLpb")
      on ReleaseLeft: ResetBit("SCLpb")
   RoundButton "Round button_4" at 388,381 size 48x48; Text 'STL'
      on PressLeft: SetBit("STLpb")
      on ReleaseLeft: ResetBit("STLpb")
   TextField "Text field_10" at 330,296 size 130x26; Text 'Function Block'
      Visibility <- "ProgramLanguage"
   TextField "Text field_11" at 306,295 size 164x26; Text 'Structured Control'
      Visibility <- "ProgramLanguage"
   TextField "Text field_12" at 325,295 size 132x26; Text 'Statement List'
      Visibility <- "ProgramLanguage"
   RoundButton "Round button_5" at 34,335 size 94x94; Text 'START'
      on PressLeft: SetBit("SystemStartPb")
      on ReleaseLeft: ResetBit("SystemStartPb")
   RoundButton "Round button_6" at 153,337 size 94x94; Text 'STOP'
      on PressLeft: SetBit("SystemStopPb")
      on ReleaseLeft: ResetBit("SystemStopPb")
   IOField "I/O field_1" at 190,136 size 80x55; FormatPattern s99999
      ProcessValue <- "Current"
   TextField "Text field_13" at 104,151 size 73x24; Text 'Current:'
   TextField "Text field_14" at 278,151 size 28x24; Text 'kW'
   TextField "Text field_15" at 90,226 size 85x24; Text 'Interlock:'
   TextField "Text field_16" at 185,223 size 93x30; Text 'ENGAGED'
      Visibility <- "StationintlkEn"
   Group "Group_1" at 445,447 size 48x48
   Group "Group" at 445,447 size 48x48
      Visibility <- "FaultMode"
   TextField "Text field_18" at 291,270 size 194x19; Text 'Programming Language'
   TextField "Text field_2" at 456,462 size 25x19; Text 'OK!'
   TextField "Text field_1" at 445,461 size 47x19; Text 'Alarm!'

screen "Overview" 500x500
   Button "Button_1" at 13,455 size 80x30; TextOff 'Main'
      on Click: ActivateScreen("Status", 0)
   Button "Button_2" at 109,455 size 80x30; TextOff 'Overview'
      on Click: ActivateScreen("Overview", 0)
   Button "Button_3" at 205,455 size 80x30; TextOff 'Alarms'
      on Click: ActivateScreen("Alarms", 0)
   Button "Button_4" at 301,455 size 80x30; TextOff 'Config'
      on Click: ActivateScreen("Config", 0)
   TextField "Text field_3" at 8,8 size 154x24; Text 'System Overview'
   Group "Group_1" at 445,447 size 48x48
   Group "Group" at 445,447 size 48x48
      Visibility <- "FaultMode"
   GraphicView "Graphic view_1" at -13,32 size 520x324; Picture "System2_1"
   IOField "I/O field_1" at 8,332 size 63x38; FormatPattern 99999999
      ProcessValue <- "BafflePct"
   TextField "Text field_4" at 13,370 size 60x19; Text 'Baffle %'
   IOField "I/O field_2" at 238,332 size 63x38; FormatPattern 99999999
      ProcessValue <- "RPM"
   TextField "Text field_5" at 251,370 size 31x19; Text 'RPM'
   IOField "I/O field_3" at 189,122 size 63x38; FormatPattern 99999999
      ProcessValue <- "VFDpct"
   TextField "Text field_6" at 178,160 size 87x19; Text 'Oil Pump %'
   Group "Group_2" at 251,64 size 148x32
      Visibility <- "StationintlkEn"
   Group "Group_3" at 251,64 size 148x32
      Visibility <- "StationintlkEn"
   Group "Group_4" at 343,334 size 148x32
      Visibility <- "BrakeEn"
   Group "Group_5" at 343,334 size 148x32
      Visibility <- "BrakeEn"
   Group "Group_6" at 20,47 size 48x48
      Visibility <- "EStopAlarm"
   Group "Group_7" at 68,47 size 48x48
      Visibility <- "BrakeFailureAlarm"
   Group "Group_8" at 116,47 size 48x48
      Visibility <- "HighOilTempAlarm"
   Group "Group_9" at 20,95 size 48x48
      Visibility <- "HighOilFlowAlarm"
   Group "Group_10" at 68,95 size 48x48
      Visibility <- "LowOilFlowAlarm"
   Group "Group_11" at 116,95 size 48x48
      Visibility <- "OvercurrentAlarm"
   Group "Group_12" at 20,45 size 147x102
      Visibility <- "FaultMode"
   TextField "Text field_18" at 131,406 size 134x38; Text 'Idle Mode'
      Visibility <- "ModeInt"
   TextField "Text field_19" at 69,406 size 196x38; Text 'Warmup Mode'
      Visibility <- "ModeInt"
   TextField "Text field_20" at 72,406 size 193x38; Text 'Stabilize Mode'
      Visibility <- "ModeInt"
   TextField "Text field_21" at 36,406 size 229x38; Text 'Generation Mode'
      Visibility <- "ModeInt"
   TextField "Text field_22" at 53,406 size 212x38; Text 'Cooldown Mode'
      Visibility <- "ModeInt"
   Button "Button_5" at 403,388 size 80x30; TextOff 'Exit App'
      on Click: StopRuntime(0)
   IOField "I/O field_4" at 123,334 size 63x38; FormatPattern 99999999
      ProcessValue <- "OilTemp"
   TextField "Text field_23" at 120,372 size 66x19; Text 'Oil Temp'
   IOField "I/O field_5" at 318,391 size 63x38; FormatPattern 99999999
      ProcessValue <- "Current"
   TextField "Text field_24" at 336,429 size 22x19; Text 'kW'
   TextField "Text field_2" at 456,462 size 25x19; Text 'OK!'
   TextField "Text field_1" at 445,461 size 47x19; Text 'Alarm!'
   TextField "Text field_8" at 363,340 size 106x19; Text 'Brake Released'
   TextField "Text field_7" at 360,339 size 109x19; Text 'Brake Engaged!'
   TextField "Text field_10" at 262,70 size 128x19; Text 'Interlock Engaged'
   TextField "Text field_9" at 279,69 size 91x19; Text 'No Interlock!'
   TextField "Text field_11" at 23,61 size 41x19; Text 'EStop'
   TextField "Text field_12" at 73,61 size 39x19; Text 'Brake'
   TextField "Text field_13" at 120,61 size 41x19; Text 'Temp'
   TextField "Text field_14" at 25,111 size 38x17; Text 'HiFlow'
   TextField "Text field_15" at 71,111 size 42x17; Text 'LoFlow'
   TextField "Text field_16" at 129,111 size 22x19; Text 'kW'
   TextField "Text field_17" at 48,81 size 97x24; Text 'No Alarms.'

screen "Alarms" 500x500
   Button "Button_1" at 13,455 size 80x30; TextOff 'Main'
      on Click: ActivateScreen("Status", 0)
   Button "Button_2" at 109,455 size 80x30; TextOff 'Overview'
      on Click: ActivateScreen("Overview", 0)
   Button "Button_3" at 205,455 size 80x30; TextOff 'Alarms'
      on Click: ActivateScreen("Alarms", 0)
   Button "Button_4" at 301,455 size 80x30; TextOff 'Config'
      on Click: ActivateScreen("Config", 0)
   TextField "Text field_3" at 8,8 size 174x24; Text 'Alarm Management'
   AlarmControl "Alarm view_1" at 15,44 size 472x254
   RoundButton "Round button_1" at 264,347 size 75x75; Text 'Silence'
      on PressLeft: SetBit("AlarmSilence")
      on ReleaseLeft: ResetBit("AlarmSilence")
   RoundButton "Round button_2" at 352,347 size 75x75; Text 'Reset'
      on PressLeft: SetBit("AlarmReset")
      on ReleaseLeft: ResetBit("AlarmReset")
   TextField "Text field_4" at 284,316 size 116x22; Text 'Alarm Controls'
   Group "Group_2" at 43,333 size 48x48
      Visibility <- "EStopAlarm"
   Group "Group_3" at 91,333 size 48x48
      Visibility <- "BrakeFailureAlarm"
   Group "Group_4" at 139,333 size 48x48
      Visibility <- "HighOilTempAlarm"
   Group "Group_5" at 43,381 size 48x48
      Visibility <- "HighOilFlowAlarm"
   Group "Group_6" at 91,381 size 48x48
      Visibility <- "LowOilFlowAlarm"
   Group "Group_7" at 139,381 size 48x48
      Visibility <- "OvercurrentAlarm"
   Group "Group_8" at 43,331 size 147x102
      Visibility <- "FaultMode"
   Group "Group_1" at 445,447 size 48x48
   Group "Group" at 445,447 size 48x48
      Visibility <- "FaultMode"
   TextField "Text field_5" at 46,347 size 41x19; Text 'EStop'
   TextField "Text field_6" at 96,347 size 39x19; Text 'Brake'
   TextField "Text field_7" at 143,347 size 41x19; Text 'Temp'
   TextField "Text field_8" at 48,397 size 38x17; Text 'HiFlow'
   TextField "Text field_9" at 94,397 size 42x17; Text 'LoFlow'
   TextField "Text field_10" at 152,397 size 22x19; Text 'kW'
   TextField "Text field_11" at 71,367 size 97x24; Text 'No Alarms.'
   TextField "Text field_2" at 456,462 size 25x19; Text 'OK!'
   TextField "Text field_1" at 445,461 size 47x19; Text 'Alarm!'

screen "Config" 500x500
   TextField "Text field_2" at 456,462 size 25x19; Text 'OK!'
   Group "Group_1" at 445,447 size 48x48
   Button "Button_1" at 13,455 size 80x30; TextOff 'Main'
      on Click: ActivateScreen("Status", 0)
   Button "Button_2" at 109,455 size 80x30; TextOff 'Overview'
      on Click: ActivateScreen("Overview", 0)
   Button "Button_3" at 205,455 size 80x30; TextOff 'Alarms'
      on Click: ActivateScreen("Alarms", 0)
   Button "Button_4" at 301,455 size 80x30; TextOff 'Config'
      on Click: ActivateScreen("Config", 0)
   Group "Group" at 445,447 size 48x48
      Visibility <- "FaultMode"
   TextField "Text field_3" at 8,8 size 125x24; Text 'Configuration'
   Group "Group_3" at 327,209 size 166x237
   Group "Group_5" at 11,404 size 289x40
   TextField "Text field_21" at 387,11 size 98x19; Text 'HOA Controls'
   TextField "Text field_22" at 342,35 size 38x17; Text 'Horn'
   TextField "Text field_23" at 336,59 size 39x17; Text 'Brake'
   TextField "Text field_24" at 317,81 size 58x17; Text 'Interlock'
   TextField "Text field_25" at 323,105 size 119x17; Text 'Baffle'
   TextField "Text field_26" at 320,156 size 90x17; Text 'Oil Pump VFD'
   Button "Button_5" at 376,34 size 24x20; TextOff 'H'
      on PressLeft: SetBit("AlarmHornHandPb")
      on ReleaseLeft: ResetBit("AlarmHornHandPb")
   Button "Button_6" at 403,34 size 24x20; TextOff 'O'
      on PressLeft: SetBit("AlarmHornOffPb")
      on ReleaseLeft: ResetBit("AlarmHornOffPb")
   Button "Button_7" at 430,34 size 24x20; TextOff 'A'
      on PressLeft: SetBit("AlarmHornAutoPb")
      on ReleaseLeft: ResetBit("AlarmHornAutoPb")
   Rectangle "Rectangle_4" at 460,34 size 25x20
      Visibility <- "AlarmHornHOA"
   Rectangle "Rectangle_5" at 460,34 size 25x20
      Visibility <- "AlarmHornHOA"
   Rectangle "Rectangle_6" at 460,34 size 25x20
      Visibility <- "AlarmHornHOA"
   Rectangle "Rectangle_7" at 460,57 size 25x20
      Visibility <- "BrakeHOA"
   Rectangle "Rectangle_8" at 460,57 size 25x20
      Visibility <- "BrakeHOA"
   Rectangle "Rectangle_9" at 461,57 size 25x20
      Visibility <- "BrakeHOA"
   Rectangle "Rectangle_10" at 460,80 size 25x20
      Visibility <- "StationintlkHOA"
   Rectangle "Rectangle_11" at 460,80 size 25x20
      Visibility <- "StationintlkHOA"
   Rectangle "Rectangle_12" at 461,80 size 25x20
      Visibility <- "StationintlkHOA"
   Rectangle "Rectangle_13" at 393,131 size 25x20
      Visibility <- "BaffleHOA"
   Rectangle "Rectangle_14" at 393,131 size 25x20
      Visibility <- "BaffleHOA"
   Rectangle "Rectangle_15" at 394,131 size 25x20
      Visibility <- "BaffleHOA"
   Rectangle "Rectangle_16" at 392,179 size 25x20
      Visibility <- "VFDhoa"
   Rectangle "Rectangle_17" at 392,179 size 25x20
      Visibility <- "VFDhoa"
   Rectangle "Rectangle_18" at 393,179 size 25x20
      Visibility <- "VFDhoa"
   Button "Button_8" at 376,57 size 24x20; TextOff 'H'
      on PressLeft: SetBit("BrakeHandPb")
      on ReleaseLeft: ResetBit("BrakeHandPb")
   Button "Button_9" at 403,57 size 24x20; TextOff 'O'
      on PressLeft: SetBit("BrakeOffPb")
      on ReleaseLeft: ResetBit("BrakeOffPb")
   Button "Button_10" at 430,57 size 24x20; TextOff 'A'
      on PressLeft: SetBit("BrakeAutoPb")
      on ReleaseLeft: ResetBit("BrakeAutoPb")
   Button "Button_11" at 376,80 size 24x20; TextOff 'H'
      on PressLeft: SetBit("StationintlkHandPb")
      on ReleaseLeft: ResetBit("StationintlkHandPb")
   Button "Button_12" at 403,80 size 24x20; TextOff 'O'
      on PressLeft: SetBit("StationintlkOffPb")
      on ReleaseLeft: ResetBit("StationintlkOffPb")
   Button "Button_13" at 430,80 size 24x20; TextOff 'A'
      on PressLeft: SetBit("StationintlkAutoPb")
      on ReleaseLeft: ResetBit("StationintlkAutoPb")
   Button "Button_14" at 312,131 size 24x20; TextOff 'H'
      on PressLeft: SetBit("BaffleHandPb")
      on ReleaseLeft: ResetBit("BaffleHandPb")
   Button "Button_15" at 339,131 size 24x20; TextOff 'O'
      on PressLeft: SetBit("BaffleOffPb")
      on ReleaseLeft: ResetBit("BaffleOffPb")
   Button "Button_16" at 366,131 size 24x20; TextOff 'A'
      on PressLeft: SetBit("BaffleAutoPb")
      on ReleaseLeft: ResetBit("BaffleAutoPb")
   Button "Button_17" at 312,179 size 24x20; TextOff 'H'
      on PressLeft: SetBit("VFDhandPb")
      on ReleaseLeft: ResetBit("VFDhandPb")
   Button "Button_18" at 339,179 size 24x20; TextOff 'O'
      on PressLeft: SetBit("VFDoffPb")
      on ReleaseLeft: ResetBit("VFDoffPb")
   Button "Button_19" at 366,179 size 24x20; TextOff 'A'
      on PressLeft: SetBit("VFDautoPb")
      on ReleaseLeft: ResetBit("VFDautoPb")
   IOField "I/O field_16" at 423,119 size 64x32; FormatPattern s999999999.999
      ProcessValue <- "BaffleManualSp"
   IOField "I/O field_17" at 423,167 size 64x32; FormatPattern s999999999.999
      ProcessValue <- "VFDmanualSp"
   TextField "Text field_27" at 432,107 size 53x17; Text 'Manual Sp'
   TextField "Text field_28" at 432,155 size 53x17; Text 'Manual Sp'
   Group "Group_2" at 8,34 size 186x365
   TextField "Text field_1" at 445,461 size 47x19; Text 'Alarm!'
   IOField "I/O field_1" at 436,240 size 49x26; FormatPattern s99999
      ProcessValue <- "WarmupOilTemp"
   TextField "Text field_4" at 374,213 size 104x19; Text 'Process Values'
   TextField "Text field_5" at 340,242 size 93x17; Text 'Warmup Temp'
   TextField "Text field_6" at 340,277 size 92x17; Text 'Warmup Delay'
   TextField "Text field_7" at 350,311 size 82x17; Text 'Current (kW)'
   TextField "Text field_8" at 342,344 size 97x17; Text 'Stabilize Delay'
   TextField "Text field_9" at 332,378 size 100x17; Text 'Cooldown Temp'
   TextField "Text field_10" at 333,412 size 99x17; Text 'Cooldown Delay'
   IOField "I/O field_2" at 436,274 size 49x26; FormatPattern s99999
      ProcessValue <- "WarmUpDelay"
   IOField "I/O field_3" at 436,308 size 49x26; FormatPattern s99999
      ProcessValue <- "CurrentSp"
   IOField "I/O field_4" at 436,342 size 49x26; FormatPattern s99999
      ProcessValue <- "StabilizeDelay"
   IOField "I/O field_5" at 436,376 size 49x26; FormatPattern s99999
      ProcessValue <- "CooldownOilTemp"
   IOField "I/O field_6" at 436,410 size 49x26; FormatPattern s99999
      ProcessValue <- "CooldownDelay"
   IOField "I/O field_7" at 136,65 size 49x26; FormatPattern s99999
      ProcessValue <- "BrakeFailureDelay"
   TextField "Text field_11" at 88,38 size 94x19; Text 'Alarm Values'
   TextField "Text field_12" at 13,68 size 123x17; Text 'Brake Failure Delay'
   TextField "Text field_13" at 34,99 size 101x17; Text 'Overspeed RPM'
   TextField "Text field_14" at 27,127 size 107x17; Text 'Overspeed Delay'
   TextField "Text field_15" at 14,156 size 119x17; Text 'Overtemp Degrees'
   TextField "Text field_16" at 30,185 size 105x17; Text 'Overtemp Delay'
   IOField "I/O field_8" at 136,95 size 49x26; FormatPattern s99999
      ProcessValue <- "OverspeedSp"
   IOField "I/O field_9" at 136,124 size 49x26; FormatPattern s99999
      ProcessValue <- "OverspeedDelay"
   IOField "I/O field_10" at 136,153 size 49x26; FormatPattern s99999
      ProcessValue <- "HighOilTempSp"
   IOField "I/O field_11" at 136,183 size 49x26; FormatPattern s99999
      ProcessValue <- "HighOilTempDelay"
   TextField "Text field_17" at 51,215 size 84x17; Text 'Lo Flow GPM'
   TextField "Text field_18" at 42,245 size 92x17; Text 'Lo Flow Delay'
   TextField "Text field_19" at 51,275 size 84x17; Text 'Hi Flow GPM'
   TextField "Text field_20" at 46,305 size 87x17; Text 'Hi Flow Delay'
   IOField "I/O field_12" at 136,211 size 49x26; FormatPattern s99999
      ProcessValue <- "LowOilFlowSp"
   IOField "I/O field_13" at 136,241 size 49x26; FormatPattern s99999
      ProcessValue <- "LowOilFlowDelay"
   IOField "I/O field_14" at 136,271 size 49x26; FormatPattern s99999
      ProcessValue <- "HighOilFlowSp"
   IOField "I/O field_15" at 136,301 size 49x26; FormatPattern s99999
      ProcessValue <- "HighOilFlowDelay"
   TextField "Text field_33" at 30,335 size 102x17; Text 'Overcurrent kW'
   TextField "Text field_34" at 16,364 size 120x17; Text 'Overcurrent Delay'
   IOField "I/O field_21" at 136,332 size 49x26; FormatPattern s99999
      ProcessValue <- "OverCurrentSp"
   IOField "I/O field_22" at 136,362 size 49x26; FormatPattern s99999
      ProcessValue <- "OvercurrentDelay"
   IOField "I/O field_18" at 83,404 size 49x26; FormatPattern s99999
      ProcessValue <- "HM_Days"
   TextField "Text field_29" at 11,406 size 75x17; Text 'Hourmeter'
   Button "Button_20" at 251,404 size 49x25; TextOff 'RESET'
      on PressLeft: SetBit("HM_ResetPb")
      on ReleaseLeft: ResetBit("HM_ResetPb")
   IOField "I/O field_19" at 137,404 size 49x26; FormatPattern s99999
      ProcessValue <- "HM_Hours"
   IOField "I/O field_20" at 191,404 size 49x26; FormatPattern s99999
      ProcessValue <- "HM_Minutes"
   TextField "Text field_30" at 93,427 size 43x17; Text 'Days'
   TextField "Text field_31" at 202,427 size 43x17; Text 'Mins'
   TextField "Text field_32" at 143,427 size 43x17; Text 'Hours'
*)